TYPE csp_transfer_accumulator_accU_depth_enum :
(
	CSP_TRANSFER_ACCUMULATOR_ACCU_DEPTH_STATUS_NOT_INITIALIZED 									:= 0,
	CSP_TRANSFER_ACCUMULATOR_ACCU_DEPTH_STATUS_DISABLED 										:= 10,
	CSP_TRANSFER_ACCUMULATOR_ACCU_DEPTH_STATUS_POSITION_CHECK									:= 20,
	CSP_TRANSFER_ACCUMULATOR_ACCU_DEPTH_STATUS_ENABLE_REQUEST 									:= 30,
	CSP_TRANSFER_ACCUMULATOR_ACCU_DEPTH_STATUS_ENABLED 											:= 40,
	CSP_TRANSFER_ACCUMULATOR_ACCU_DEPTH_STATUS_GEAR_REQUEST										:= 50,
	CSP_TRANSFER_ACCUMULATOR_ACCU_DEPTH_STATUS_GEARING											:= 60,
	CSP_TRANSFER_ACCUMULATOR_ACCU_DEPTH_STATUS_GEARED											:= 70,
	CSP_TRANSFER_ACCUMULATOR_ACCU_DEPTH_STATUS_MOVING											:= 80,
	CSP_TRANSFER_ACCUMULATOR_ACCU_DEPTH_STATUS_DISENGAGE_REQUEST								:= 90,
	CSP_TRANSFER_ACCUMULATOR_ACCU_DEPTH_STATUS_DISENGAGING										:= 100,
	CSP_TRANSFER_ACCUMULATOR_ACCU_DEPTH_STATUS_STOP_REQUEST 									:= 110,
	CSP_TRANSFER_ACCUMULATOR_ACCU_DEPTH_STATUS_DISABLE_REQUEST 									:= 120,
	CSP_TRANSFER_ACCUMULATOR_ACCU_DEPTH_STATUS_DISABLING 										:= 130
) := CSP_TRANSFER_ACCUMULATOR_ACCU_DEPTH_STATUS_NOT_INITIALIZED;
END_TYPE

(* stored: Version 1.1.0.1, ProductVersion 3.1.4024.3
   DUT csp_transfer_accumulator_accU_depth_enum: Id {13049e30-2df9-47e4-af28-2651f754e1e2} *)
